// TIA Portal project "Confirm v7_V17" (V17)

(* hardware
DEVICE "S71500/ET200MP station_1"  S7-1500 station
   slot 0: "Rail_0"  Rack  6ES7 590-1***0-0AA0
   slot 1: "PLC1"  CPU 1512C-1 PN  6ES7 512-1CK01-0AB0  V2.5
      slot 3: "CPU display_1"  6ES7591-1AA00-0AA0
      slot 32768: "PROFINET interface_1"  X1
         slot 32769: "Port_1"  X1 P1
         slot 32770: "Port_2"  X1 P2
DEVICE "S71500/ET200MP station_2"  S7-1500 station
   slot 0: "Rail_0"  Rack  6ES7 590-1***0-0AA0
   slot 1: "PLC_2"  CPU 1512C-1 PN  6ES7 512-1CK01-0AB0  V2.5
      slot 3: "CPU display_1"  6ES7591-1AA00-0AA0
      slot 32768: "PROFINET interface_1"  X1
         slot 32769: "Port_1"  X1 P1
         slot 32770: "Port_2"  X1 P2
*)

// ===== PLC "PLC1"  CPU 1512C-1 PN =====

VAR_GLOBAL   // PLC tag table "Default tag table"
   "START" AT %I10.0 : Bool;
   "STOP" AT %I10.1 : Bool;
   "MANUAL" AT %I10.2 : Bool;
   "RESET" AT %I10.3 : Bool;
   "START LED" AT %Q4.0 : Bool;
   "RESET LED" AT %Q4.1 : Bool;
   "Q1 LED" AT %Q4.2 : Bool;
   "Q2 LED" AT %Q4.3 : Bool;
   "extend_feed_cyl" AT %Q4.4 : Bool;
   "Tag_2" AT %QB4 : Byte;
   "reset_timer_delay_bit" AT %M0.1 : Bool;
   "convoy_motor" AT %Q4.5 : Bool;
   "Stopper" AT %Q4.6 : Bool;
   "Tag_7" AT %I0.0 : Bool;
   "Tag_8" AT %M2.0 : Bool;
   "Tag_9" AT %M9.4 : Bool;
   "O/P command to Robot Arm" AT %Q5.0 : Bool;
   "O/P command to NX" AT %Q5.4 : Bool;
   "robot return to home" AT %Q6.0 : Bool;
   "conveyor 3" AT %Q6.4 : Bool;
   "Tag_14" AT %Q7.0 : Bool;
   "Tag_15" AT %Q7.7 : Bool;
   "Tag_16" AT %Q7.4 : Bool;
   "Tag_17" AT %QD4 : DWord;
   "start_comparison" AT %M0.2 : Bool;
   "stop_comparison" AT %M0.3 : Bool;
   "obj_pres(Dissuse_sensor)" AT %I10.5 : Bool;
   "Metal(Ind_sensor)" AT %I10.6 : Bool;
   "color_sensor" AT %I10.7 : Bool;
   "feed_cyl_extended" AT %I11.0 : Bool;
   "feed_photo_sensor" AT %I0.1 : Bool;
   "count_down_bit" AT %Q10.6 : Bool;
   "r_bit2" AT %M0.5 : Bool;
   "power_on_mem" AT %M0.0 : Bool;
   "manual_output" AT %Q15.0 : Bool;
   "reflective_light_sensor" AT %I11.1 : Bool;
   "chute_full_notification" AT %Q5.6 : Bool;
   "wkpiece in  conveyor 3" AT %I11.2 : Bool;
END_VAR

DATA_BLOCK "Data_block_1"   // DB1
{ S7_Optimized_Access := 'FALSE' }
VERSION : 0.1
   VAR
      start_bit : Bool;
      stop_bit : Bool;
      reset_bit : Bool;
      manual_set_bit : Bool;
      power_on_mem : Bool;
      "system_active?" : Bool;
      process_no : Word;
      time_preset : Time := T#2_500MS;
      monitering_time : Time;
   END_VAR
BEGIN
END_DATA_BLOCK

// folder: System blocks/Program resources

DATA_BLOCK "reset_button_timer1"   // DB2
{ S7_Optimized_Access := 'TRUE' }
AUTHOR : Simatic
FAMILY : IEC
NAME : IEC_TMR
VERSION : 1.0
// stored: InstanceOfName IEC_TIMER
"IEC_TIMER"
BEGIN
END_DATA_BLOCK

DATA_BLOCK "Timer_for_met_sensor"   // DB3
{ S7_Optimized_Access := 'TRUE' }
AUTHOR : Simatic
FAMILY : IEC
NAME : IEC_TMR
VERSION : 1.0
// stored: InstanceOfName IEC_TIMER
"IEC_TIMER"
BEGIN
END_DATA_BLOCK

DATA_BLOCK "reset_button_timer2"   // DB4
{ S7_Optimized_Access := 'TRUE' }
AUTHOR : Simatic
FAMILY : IEC
NAME : IEC_TMR
VERSION : 1.0
// stored: InstanceOfName IEC_TIMER
"IEC_TIMER"
BEGIN
END_DATA_BLOCK

DATA_BLOCK "wait_time1"   // DB5
{ S7_Optimized_Access := 'TRUE' }
AUTHOR : Simatic
FAMILY : IEC
NAME : IEC_TMR
VERSION : 1.0
// stored: InstanceOfName IEC_TIMER
"IEC_TIMER"
BEGIN
END_DATA_BLOCK

DATA_BLOCK "Count_for_unwanted"   // DB6
{ S7_Optimized_Access := 'TRUE' }
AUTHOR : Simatic
FAMILY : IEC
NAME : CNTR
VERSION : 1.0
// stored: InstanceOfName IEC_COUNTER
"IEC_COUNTER"
BEGIN
END_DATA_BLOCK

DATA_BLOCK "counter_wanted"   // DB7
{ S7_Optimized_Access := 'TRUE' }
AUTHOR : Simatic
FAMILY : IEC
NAME : CNTR
VERSION : 1.0
// stored: InstanceOfName IEC_COUNTER
"IEC_COUNTER"
BEGIN
END_DATA_BLOCK

DATA_BLOCK "Robot_arm_waiting_timer"   // DB8
{ S7_Optimized_Access := 'TRUE' }
AUTHOR : Simatic
FAMILY : IEC
NAME : IEC_TMR
VERSION : 1.0
// stored: InstanceOfName IEC_TIMER
"IEC_TIMER"
BEGIN
END_DATA_BLOCK

DATA_BLOCK "chute_full_timer"   // DB9
{ S7_Optimized_Access := 'TRUE' }
AUTHOR : Simatic
FAMILY : IEC
NAME : IEC_TMR
VERSION : 1.0
// stored: InstanceOfName IEC_TIMER
"IEC_TIMER"
BEGIN
END_DATA_BLOCK

DATA_BLOCK "reset_time_latch_countdown1"   // DB10
{ S7_Optimized_Access := 'TRUE' }
AUTHOR : Simatic
FAMILY : IEC
NAME : IEC_TMR
VERSION : 1.0
// stored: InstanceOfName IEC_TIMER
"IEC_TIMER"
BEGIN
END_DATA_BLOCK

// folder: (top level)

FUNCTION "Auto_Mode" : Void   // FC1, LAD
{ S7_Optimized_Access := 'TRUE' }
VERSION : 0.1
   VAR_TEMP   // added for the SCL form of the ladder/FBD networks
      _w1 : Bool;
   END_VAR
BEGIN

REGION Network 1: Detection of material at entry
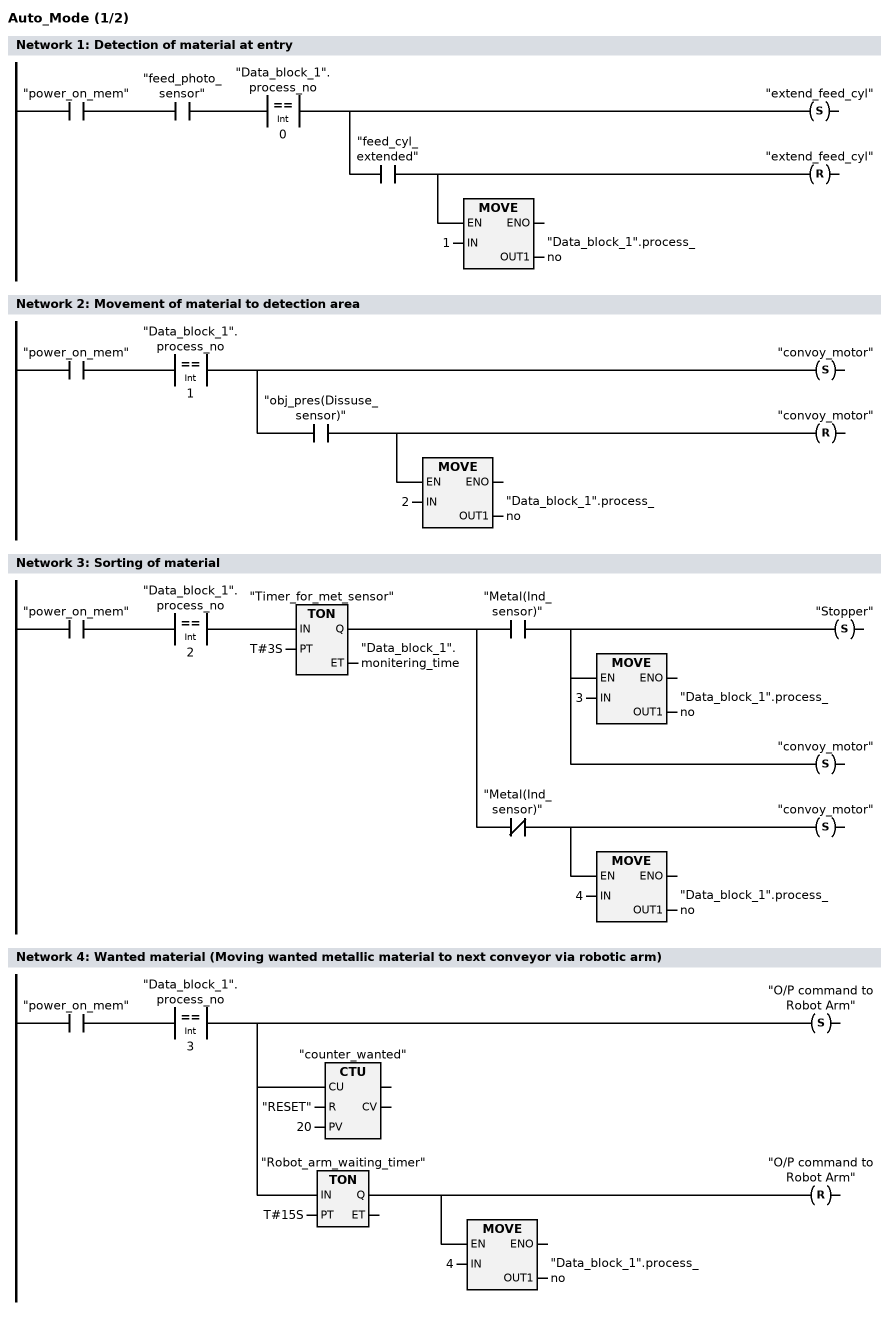
   RUNG wire#powerrail
      Contact( "power_on_mem" )
      Contact( "feed_photo_sensor" )
      { S7_Templates := "SrcType := Int" } EQ_Contact(in1 := "Data_block_1".process_no, in2 := 0)
      wire#w1
      S_Coil( "extend_feed_cyl" )
   END_RUNG
   RUNG wire#w1
      Contact( "feed_cyl_extended" )
      wire#w2
      R_Coil( "extend_feed_cyl" )
   END_RUNG
   RUNG wire#w2
      Move(in := 1, out1 => "Data_block_1".process_no)
   END_RUNG
   // the same network as SCL:
   #_w1 := "power_on_mem" AND "feed_photo_sensor" AND ("Data_block_1".process_no = 0);
   IF #_w1 THEN "extend_feed_cyl" := TRUE; END_IF;
   IF #_w1 AND "feed_cyl_extended" THEN
       "extend_feed_cyl" := FALSE;
       "Data_block_1".process_no := 1;
   END_IF;
END_REGION

REGION Network 2: Movement of material to detection area
   RUNG wire#powerrail
      Contact( "power_on_mem" )
      { S7_Templates := "SrcType := Int" } EQ_Contact(in1 := "Data_block_1".process_no, in2 := 1)
      wire#w1
      S_Coil( "convoy_motor" )
   END_RUNG
   RUNG wire#w1
      Contact( "obj_pres(Dissuse_sensor)" )
      wire#w2
      R_Coil( "convoy_motor" )
   END_RUNG
   RUNG wire#w2
      Move(in := 2, out1 => "Data_block_1".process_no)
   END_RUNG
   // the same network as SCL:
   #_w1 := "power_on_mem" AND ("Data_block_1".process_no = 1);
   IF #_w1 THEN "convoy_motor" := TRUE; END_IF;
   IF #_w1 AND "obj_pres(Dissuse_sensor)" THEN
       "convoy_motor" := FALSE;
       "Data_block_1".process_no := 2;
   END_IF;
END_REGION

REGION Network 3: Sorting of material
   "Timer_for_met_sensor".TON(IN := "power_on_mem" AND ("Data_block_1".process_no = 2),
                           PT := T#3S,
                           ET => "Data_block_1".monitering_time);
   IF "Timer_for_met_sensor".Q AND "Metal(Ind_sensor)" THEN
       "Stopper" := TRUE;
       "Data_block_1".process_no := 3;
       "convoy_motor" := TRUE;
   END_IF;
   IF "Timer_for_met_sensor".Q AND NOT "Metal(Ind_sensor)" THEN
       "convoy_motor" := TRUE;
       "Data_block_1".process_no := 4;
   END_IF;
END_REGION

REGION Network 4: Wanted material (Moving wanted metallic material to next conveyor via robotic arm)
   #_w1 := "power_on_mem" AND ("Data_block_1".process_no = 3);
   IF #_w1 THEN "O/P command to Robot Arm" := TRUE; END_IF;
   "counter_wanted".CTU(CU := #_w1, R := "RESET", PV := 20);
   "Robot_arm_waiting_timer".TON(IN := #_w1, PT := T#15S);
   IF "Robot_arm_waiting_timer".Q THEN
       "O/P command to Robot Arm" := FALSE;
       "Data_block_1".process_no := 4;
   END_IF;
END_REGION

REGION Network 5: Wanted metallic material received
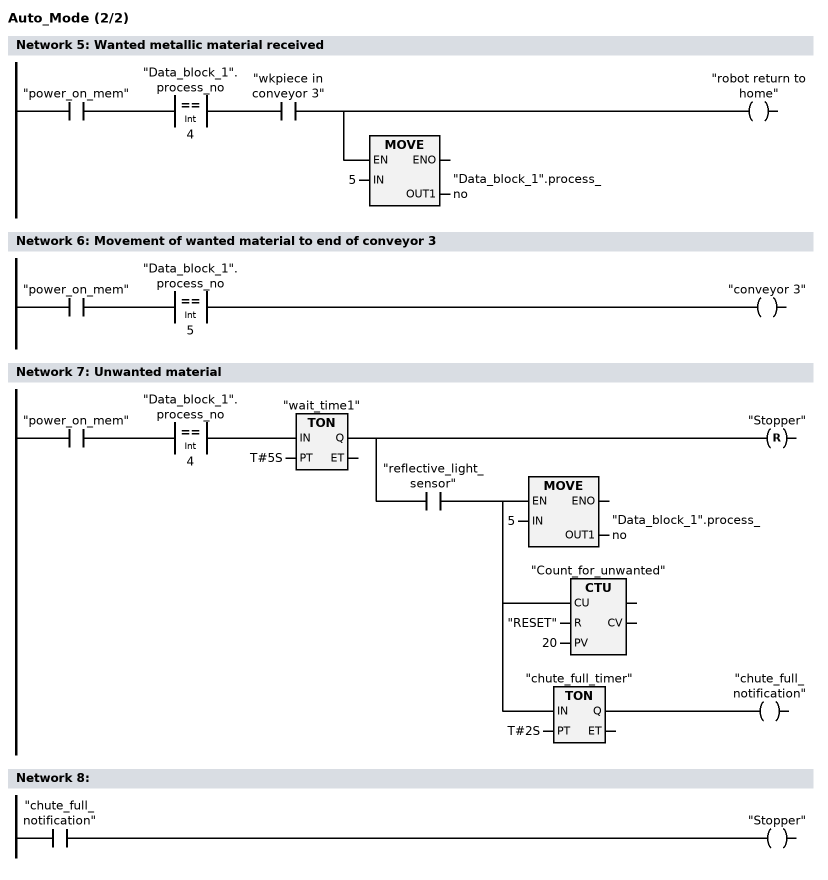
   RUNG wire#powerrail
      Contact( "power_on_mem" )
      { S7_Templates := "SrcType := Int" } EQ_Contact(in1 := "Data_block_1".process_no, in2 := 4)
      Contact( "wkpiece in  conveyor 3" )
      wire#w1
      Coil( "robot return to home" )
   END_RUNG
   RUNG wire#w1
      Move(in := 5, out1 => "Data_block_1".process_no)
   END_RUNG
   // the same network as SCL:
   "robot return to home" := "power_on_mem" AND ("Data_block_1".process_no = 4) AND "wkpiece in  conveyor 3";
   IF "robot return to home" THEN "Data_block_1".process_no := 5; END_IF;
END_REGION

REGION Network 6: Movement of wanted material to end of conveyor 3
   RUNG wire#powerrail
      Contact( "power_on_mem" )
      { S7_Templates := "SrcType := Int" } EQ_Contact(in1 := "Data_block_1".process_no, in2 := 5)
      Coil( "conveyor 3" )
   END_RUNG
   // the same network as SCL:
   "conveyor 3" := "power_on_mem" AND ("Data_block_1".process_no = 5);
END_REGION

REGION Network 7: Unwanted material
   "wait_time1".TON(IN := "power_on_mem" AND ("Data_block_1".process_no = 4), PT := T#5S);
   IF "wait_time1".Q THEN "Stopper" := FALSE; END_IF;
   #_w1 := "wait_time1".Q AND "reflective_light_sensor";
   IF #_w1 THEN "Data_block_1".process_no := 5; END_IF;
   "Count_for_unwanted".CTU(CU := #_w1, R := "RESET", PV := 20);
   "chute_full_timer".TON(IN := #_w1, PT := T#2S);
   "chute_full_notification" := "chute_full_timer".Q;
END_REGION

REGION Network 8
   RUNG wire#powerrail
      Contact( "chute_full_notification" )
      Coil( "Stopper" )
   END_RUNG
   // the same network as SCL:
   "Stopper" := "chute_full_notification";
END_REGION
END_FUNCTION

FUNCTION "Manual_Mode" : Void   // FC2, LAD
{ S7_Optimized_Access := 'TRUE' }
VERSION : 0.1
BEGIN
END_FUNCTION

ORGANIZATION_BLOCK "Main"   // OB1, LAD, ProgramCycle
TITLE = "Main Program Sweep (Cycle)"
{ S7_Optimized_Access := 'TRUE' }
VERSION : 0.1
   VAR_INPUT
      Initial_Call : Bool;   // Initial call of this OB
      Remanence : Bool;   // =True, if remanent data are available
   END_VAR
   VAR_TEMP   // added for the SCL form of the ladder/FBD networks
      _w1 : Bool;
      _w2 : Bool;
   END_VAR
BEGIN

REGION Network 1
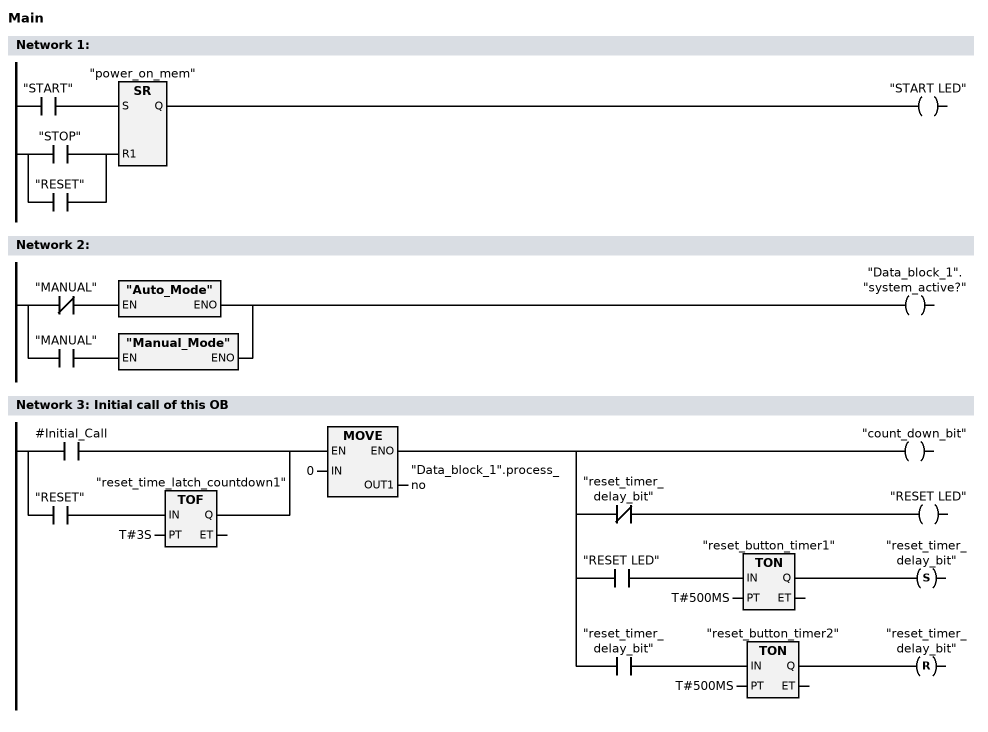
   RUNG wire#powerrail
      Contact( "START" )
      S_SR(operand := "power_on_mem", r1 := wire#w1)
      Coil( "START LED" )
   END_RUNG
   RUNG wire#powerrail
      Contact( "STOP" )
   END_RUNG wire#w1
   RUNG wire#powerrail
      Contact( "RESET" )
   END_RUNG wire#w1
   // the same network as SCL:
   IF "START" THEN
       "power_on_mem" := TRUE;   // SR flip-flop
   END_IF;
   IF "STOP" OR "RESET" THEN "power_on_mem" := FALSE; END_IF;
   "START LED" := "power_on_mem";
END_REGION

REGION Network 2
   RUNG wire#powerrail
      I_Contact( "MANUAL" )
      "Auto_Mode"()
      wire#w1
      Coil( "Data_block_1"."system_active?" )
   END_RUNG
   RUNG wire#powerrail
      Contact( "MANUAL" )
      "Manual_Mode"()
   END_RUNG wire#w1
   // the same network as SCL:
   "Auto_Mode"(EN := NOT "MANUAL", ENO => #_w1);
   "Manual_Mode"(EN := "MANUAL", ENO => #_w2);
   "Data_block_1"."system_active?" := #_w1 OR #_w2;
END_REGION

REGION Network 3: Initial call of this OB
   "reset_time_latch_countdown1".TOF(IN := "RESET", PT := T#3S);
   #_w1 := #Initial_Call OR "reset_time_latch_countdown1".Q;
   IF #_w1 THEN "Data_block_1".process_no := 0; END_IF;
   "count_down_bit" := #_w1;
   "RESET LED" := #_w1 AND NOT "reset_timer_delay_bit";
   "reset_button_timer1".TON(IN := #_w1 AND "RESET LED", PT := T#500MS);
   IF "reset_button_timer1".Q THEN "reset_timer_delay_bit" := TRUE; END_IF;
   "reset_button_timer2".TON(IN := #_w1 AND "reset_timer_delay_bit", PT := T#500MS);
   IF "reset_button_timer2".Q THEN "reset_timer_delay_bit" := FALSE; END_IF;
END_REGION
END_ORGANIZATION_BLOCK

// ===== PLC "PLC_2"  CPU 1512C-1 PN =====

VAR_GLOBAL   // PLC tag table "Default tag table"
   "start" AT %M50.0 : Bool;
   "led" AT %Q0.0 : Bool;
END_VAR

ORGANIZATION_BLOCK "Main"   // OB1, LAD, ProgramCycle
TITLE = "Main Program Sweep (Cycle)"
{ S7_Optimized_Access := 'TRUE' }
VERSION : 0.1
   VAR_INPUT
      Initial_Call : Bool;   // Initial call of this OB
      Remanence : Bool;   // =True, if remanent data are available
   END_VAR
BEGIN

REGION Network 1
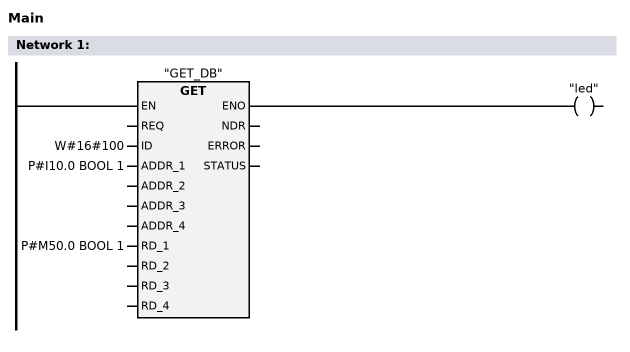
   // ENO of a box is taken as its EN; it also drops when the box reports an error
   "GET_DB"(ID := W#16#100, ADDR_1 := P#I10.0 BOOL 1, RD_1 := P#M50.0 BOOL 1);   // GET
   "led" := TRUE;
END_REGION
END_ORGANIZATION_BLOCK